// TIA Portal V17 export
// export: Created 2022-03-12T16:05:29.2173422Z, ExportSetting WithDefaults, DisplayName Totally Integrated Automation Portal, DisplayVersion V17, DisplayName TIA Portal Openness, DisplayVersion V17, DisplayName TIA Portal Version Control Interface, DisplayVersion V17, DisplayName STEP 7 Professional, DisplayVersion V17, DisplayName STEP 7 Safety, DisplayVersion V17, DisplayName WinCC Advanced / Unified PC, DisplayVersion V17
DATA_BLOCK "AlarmCfg"   // DB31600
TITLE = CPG_AlarmCfg
{ S7_Optimized_Access := 'TRUE' }
AUTHOR : tech.team.motioncontrol@siemens.com
FAMILY : CPG
VERSION : 1.0
// Support: tech.team.motioncontrol@siemens.com
// Fax: +49 (0) 9131/98-1297
// stored: AutoNumber true, DBAccessibleFromOPCUA true, DBAccessibleFromWebserver true, IsOnlyStoredInLoadMemory false, IsRetainMemResEnabled false, IsWriteProtectedInAS false, MemoryReserve 0
   VAR
      Event { ExternalAccessible := 'False'; ExternalVisible := 'False'; ExternalWritable := 'False'; S7_SetPoint := 'True'} : Array[0.."CPG_NO_OF_CFG_ALARMS_UPPER_LIM"] of "CPG_typeEventCfg";
   END_VAR
BEGIN
   // Event[0] : Alarm Test
   // Event[1] : Emergency Stop
   // Event[2] : Guard Door
   // Event[3] : Stop Command
   // Event[4] : Hold Command
   // Event[5] : Axis Error
   // Event[6] : Drive Fault
   // Event[7] : Machine Blocked
   // Event[8] : Machine Starved - No bottles
   // Event[9] : Machine Starved - No labels
   // Event[10] : Spare
   // Event[11] : Spare
   // Event[12] : Spare
   // Event[13] : Spare
   // Event[14] : Spare
   // Event[15] : Spare
   // Event[16] : Spare
   // Event[17] : Spare
   // Event[18] : Spare
   // Event[19] : Spare
   // Event[20] : Remote Stop Command
   // Event[21] : Remote Abort Command
   // Event[22] : Rmt Suspd Cmd - Blocked
   // Event[23] : Rmt Suspd Cmd - Starved
   // Event[24] : Remote Hold Cmd
   // Event[25] : Spare
   // Event[26] : Spare
   // Event[27] : Spare
   // Event[28] : Spare
   // Event[29] : Spare
   // Event[30] : Spare
   // Event[31] : Spare
   // Event[32] : Spare
   // Event[33] : Spare
   // Event[34] : Spare
   // Event[35] : Spare
   // Event[36] : Spare
   // Event[37] : Spare
   // Event[38] : Spare
   // Event[39] : Spare
   Event[0].ID := 0;
   Event[1].ID := 1;
   Event[2].ID := 4;
   Event[3].ID := 33;
   Event[4].ID := 40;
   Event[5].ID := 262;
   Event[6].ID := 261;
   Event[7].ID := 7;
   Event[8].ID := 8;
   Event[9].ID := 9;
   Event[20].ID := 41;
   Event[21].ID := 42;
   Event[22..23].ID := 43;
   Event[24].ID := 44;
   Event[1..2].value := 1;
   Event[3].value := 2;
   Event[4..5].value := 0;
   Event[6].value := 1;
   Event[7].value := 7;
   Event[8].value := 8;
   Event[9].value := 9;
   Event[20].value := 20;
   Event[21].value := 21;
   Event[22].value := 22;
   Event[23].value := 23;
   Event[24].value := 24;
   Event[38].value := 0;
   Event[0].message[0..2] := 'Alarm Test';
   Event[1].message[0] := 'E-Stop';
   Event[1].message[1] := 'Not-Halt';
   Event[1].message[2] := 'Los E-Stop';
   Event[2].message[0] := 'Guard Door';
   Event[2].message[1] := 'Schutzzaun';
   Event[2].message[2] := 'Las Guard Door';
   Event[3].message[0] := 'Stop PB';
   Event[3].message[1] := 'Stopp Taster';
   Event[3].message[2] := 'Las Stop PB';
   Event[4].message[0] := 'Hold PB';
   Event[4].message[1] := 'Hold Taster';
   Event[4].message[2] := 'Las Hold PB';
   Event[5].message[0] := 'Axis Error';
   Event[5].message[1] := 'Achsfehler';
   Event[5].message[2] := 'Las Axis Error';
   Event[6].message[0] := 'Drive Faulted';
   Event[6].message[1] := 'Antriebsfehler';
   Event[6].message[2] := 'Los Drive Faulted';
   Event[7].message[0] := 'Machine Blocked';
   Event[7].message[1] := 'Maschine blockiert';
   Event[7].message[2] := 'Los Machine Blocked';
   Event[8].message[0] := 'Starved - No botttles';
   Event[8].message[1] := 'Flaschenzufuhr leer';
   Event[8].message[2] := 'Las Starved - No botttles';
   Event[9].message[0] := 'Starved - No labels';
   Event[9].message[1] := 'Etikettenzufuhr leer';
   Event[9].message[2] := 'Las Starved - No labels';
   Event[10].message[0] := 'Spare';
   Event[10].message[1] := 'Reserve';
   Event[10].message[2] := 'Spare';
   Event[11].message[0] := 'Spare';
   Event[11].message[1] := 'Reserve';
   Event[11].message[2] := 'Spare';
   Event[12].message[0] := 'Spare';
   Event[12].message[1] := 'Reserve';
   Event[12].message[2] := 'Spare';
   Event[13].message[0] := 'Spare';
   Event[13].message[1] := 'Reserve';
   Event[13].message[2] := 'Spare';
   Event[14].message[0] := 'Spare';
   Event[14].message[1] := 'Reserve';
   Event[14].message[2] := 'Spare';
   Event[15].message[0] := 'Spare';
   Event[15].message[1] := 'Reserve';
   Event[15].message[2] := 'Spare';
   Event[16].message[0] := 'Spare';
   Event[16].message[1] := 'Reserve';
   Event[16].message[2] := 'Spare';
   Event[17].message[0] := 'Spare';
   Event[17].message[1] := 'Reserve';
   Event[17].message[2] := 'Spare';
   Event[18].message[0] := 'Spare';
   Event[18].message[1] := 'Reserve';
   Event[18].message[2] := 'Spare';
   Event[19].message[0] := 'Spare';
   Event[19].message[1] := 'Reserve';
   Event[19].message[2] := 'Spare';
   Event[20].message[0..1] := 'Remote Stop Cmd';
   Event[20].message[2] := 'Las Remote Stop Cmd';
   Event[21].message[0..1] := 'Remote Abort Cmd';
   Event[21].message[2] := 'Las Remote Abort Cmd';
   Event[22].message[0] := 'Rmt Suspd Cmd - Blocked';
   Event[22].message[1] := 'Remote Suspend Cmd - Blocked';
   Event[22].message[2] := 'Las Remote Suspd Cmd - Blocked';
   Event[23].message[0] := 'Rmt Suspd Cmd - Starved';
   Event[23].message[1] := 'Remote Suspend Cmd - Starved';
   Event[23].message[2] := 'Las Rmt Suspd Cmd - Starved';
   Event[24].message[0..1] := 'Remote Hold Cmd';
   Event[24].message[2] := 'Las Remote Hold Cmd';
   Event[25].message[0] := 'Spare';
   Event[25].message[1] := 'Reserve';
   Event[25].message[2] := 'Spare';
   Event[26].message[0] := 'Spare';
   Event[26].message[1] := 'Reserve';
   Event[26].message[2] := 'Spare';
   Event[27].message[0] := 'Spare';
   Event[27].message[1] := 'Reserve';
   Event[27].message[2] := 'Spare';
   Event[28].message[0] := 'Spare';
   Event[28].message[1] := 'Reserve';
   Event[28].message[2] := 'Spare';
   Event[29].message[0] := 'Spare';
   Event[29].message[1] := 'Reserve';
   Event[29].message[2] := 'Spare';
   Event[30].message[0] := 'Spare';
   Event[30].message[1] := 'Reserve';
   Event[30].message[2] := 'Spare';
   Event[31].message[0] := 'Spare';
   Event[31].message[1] := 'Reserve';
   Event[31].message[2] := 'Spare';
   Event[32].message[0] := 'Spare';
   Event[32].message[1] := 'Reserve';
   Event[32].message[2] := 'Spare';
   Event[33].message[0] := 'Spare';
   Event[33].message[1] := 'Reserve';
   Event[33].message[2] := 'Spare';
   Event[34].message[0] := 'Spare';
   Event[34].message[1] := 'Reserve';
   Event[34].message[2] := 'Spare';
   Event[35].message[0] := 'Spare';
   Event[35].message[1] := 'Reserve';
   Event[35].message[2] := 'Spare';
   Event[36].message[0] := 'Spare';
   Event[36].message[1] := 'Reserve';
   Event[36].message[2] := 'Spare';
   Event[37].message[0] := 'Spare';
   Event[37].message[1] := 'Reserve';
   Event[37].message[2] := 'Spare';
   Event[38].message[0] := 'Spare';
   Event[38].message[1] := 'Reserve';
   Event[38].message[2] := 'Spare';
   Event[39].message[0] := 'Spare';
   Event[39].message[1] := 'Reserve';
   Event[39].message[2] := 'Spare';
   Event[0].category := 6;
   Event[1].category := 0;   // 0 = Safety related, Coordinated fast stop
   // Event[2].category : 0 = Safety related, Coordinated fast stop
   Event[3].category := 2;   // 2 = Coordinated normal stop
   Event[4].category := 7;   // 7 = Held command
   Event[5].category := 1;   // 1 = Coordinated fast stop
   Event[6].category := 1;   // 1 = Coordinated fast stop
   Event[7].category := 8;   // 8 =Blocked, Coordinated slow stop
   Event[8].category := 9;   // 9 = Starved, Coordinated slow stop
   Event[9].category := 9;   // 9 = Starved, Coordinated slow stop
   Event[10].category := 0;   // 9 = Starved, Coordinated slow stop
   Event[11..13].category := 0;
   Event[20].category := 2;   // 2 = Coordinated normal stop
   Event[21].category := 1;   // 0 = Safety related, Coordinated fast stop
   Event[22].category := 8;   // 9 = Starved, Coordinated slow stop
   Event[23].category := 9;   // 7 = Hold, Coordinated slow stop
   Event[24].category := 7;   // 7 = Coordinated slow stop
END_DATA_BLOCK
